KUKA KRL program: Up115.src, Up115.dat

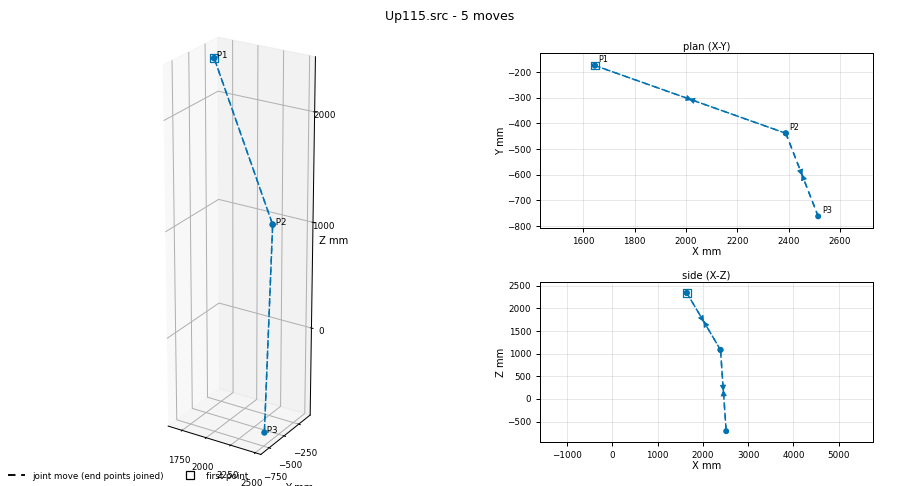
[picture p0: tool path of Up115.src, 5 of 5 moves have a stored position in this frame; points joined in program order, loops and branches not executed]
--- Up115.src ---
&ACCESS RV
&REL 2
&COMMENT Wartung Greifer 3 VW380
&PARAM DISKPATH = UPs
&PARAM TEMPLATE = C:\KRC\Roboter\Template\upvorgabe
&PARAM TPVW_VERSION = 8.1.8
&PARAM EDITMASK = Up999[1-999]
DEF UP115()
   ; FOLD UP Anfang;%{SE} %MKUKATPVW
   SPS_N=-1
   SPS_FERTIG=FALSE
   IF NOT CALLBYSELECT THEN
      INTERRUPT DECL 10 WHEN $CYCFLAG[254]==FALSE DO VW(#FB_STOP,TRUE)
      INTERRUPT ON 10
      INT10=TRUE
      VW_USR_R (#USR_INIT)
   ENDIF
   VW(#VW_INIT_UP,TRUE)
   ; ENDFOLD
   ;FOLD -- K2TUHR115425R01 Wartung Greifer VW380 -- ;%{PSE}%MKUKATPVW,%CVW_COM,%VCOMMENT,%P 1:Comment:, 2:K2TUHR115425R01 Wartung Greifer VW380
      ;FOLD {H}
         M_COMMENT("K2TUHR115425R01 Wartung Greifer VW380")
      ;ENDFOLD
   ;ENDFOLD
   ;FOLD PTP VB=100% VE=0% ACC=100% RobWzg=12 Base=0 SPSTrig=0[1/100s] P ;%{P}%MKUKATPVW,%CMOVE8,%VPTP,%P 1:1, 2: VB=, 3:100, 4:%, 5: VE=, 6:0, 7:%, 8: ACC=, 9:100, 10:%, 11: RobWzg=, 12:12, 13: Base=, 14:0, 15: SPSTrig=, 16:0, 17:[1/100s], 18: P, 19:1, 20:-1, 21:1
      ;FOLD 1: FB PSPS = EIN ;%{SE}%MKUKATPVW %CVW_SPS %VFBPSPS %P 2:FB PSPS = EIN,3:FBPSPS
      ;ENDFOLD
      ;FOLD 2: A23 = AUS ;%{SE}%MKUKATPVW %CVW_SPS %VBOASG %P 2:A23 = AUS,3:BOASG
      ;ENDFOLD
      ;FOLD 3: SPSMAKRO50 = EIN ;%{SE}%MKUKATPVW %CVW_SPS %VMAKRO %P 2:SPSMAKRO50 = EIN,3:MAKRO
      ;ENDFOLD
      ;FOLD 4: SPSMAKRO53 = EIN ;%{SE}%MKUKATPVW %CVW_SPS %VMAKRO %P 2:SPSMAKRO53 = EIN,3:MAKRO
      ;ENDFOLD
      ;FOLD 5: A42 = EIN ;%{SE}%MKUKATPVW %CVW_SPS %VBOASG %P 2:A42 = EIN,3:BOASG
      ;ENDFOLD
      ;FOLD 6: A43 = EIN ;%{SE}%MKUKATPVW %CVW_SPS %VBOASG %P 2:A43 = EIN,3:BOASG
      ;ENDFOLD
      ;FOLD 7: A44 = EIN ;%{SE}%MKUKATPVW %CVW_SPS %VBOASG %P 2:A44 = EIN,3:BOASG
      ;ENDFOLD
      ;FOLD 8: A45 = EIN ;%{SE}%MKUKATPVW %CVW_SPS %VBOASG %P 2:A45 = EIN,3:BOASG
      ;ENDFOLD
      ;FOLD 9: A47 = EIN ;%{SE}%MKUKATPVW %CVW_SPS %VBOASG %P 2:A47 = EIN,3:BOASG
      ;ENDFOLD
      ;FOLD 10: A49 = EIN ;%{SE}%MKUKATPVW %CVW_SPS %VBOASG %P 2:A49 = EIN,3:BOASG
      ;ENDFOLD
      ;FOLD 11: A52 = EIN ;%{SE}%MKUKATPVW %CVW_SPS %VBOASG %P 2:A52 = EIN,3:BOASG
      ;ENDFOLD
      ;FOLD 12: A54 = EIN ;%{SE}%MKUKATPVW %CVW_SPS %VBOASG %P 2:A54 = EIN,3:BOASG
      ;ENDFOLD
      ;FOLD 13: A75 = EIN ;%{SE}%MKUKATPVW %CVW_SPS %VBOASG %P 2:A75 = EIN,3:BOASG
      ;ENDFOLD
      ;FOLD 14: A76 = EIN ;%{SE}%MKUKATPVW %CVW_SPS %VBOASG %P 2:A76 = EIN,3:BOASG
      ;ENDFOLD
      ;FOLD 15: A79 = EIN ;%{SE}%MKUKATPVW %CVW_SPS %VBOASG %P 2:A79 = EIN,3:BOASG
      ;ENDFOLD
      ;FOLD 16: A80 = EIN ;%{SE}%MKUKATPVW %CVW_SPS %VBOASG %P 2:A80 = EIN,3:BOASG
      ;ENDFOLD
      ;FOLD 17: WARTE BIS M13 & M78 ;%{SE}%MKUKATPVW %CVW_SPS %VWBOASG %P 2:WARTE BIS M13 & M78,3:WBOASG
      ;ENDFOLD
      ;FOLD 18: F1 = EIN ;%{SE}%MKUKATPVW %CVW_SPS %VBOASG %P 2:F1 = EIN,3:BOASG
      ;ENDFOLD
      ;FOLD 19: F2 = EIN ;%{SE}%MKUKATPVW %CVW_SPS %VBOASG %P 2:F2 = EIN,3:BOASG
      ;ENDFOLD
      ;FOLD 20: SPSMAKRO342 = M13 ;%{SE}%MKUKATPVW %CVW_SPS %VMAKRO %P 2:SPSMAKRO342 = M13,3:MAKRO
      ;ENDFOLD
      ;FOLD 21: SPSMAKRO340 = EIN ;%{SE}%MKUKATPVW %CVW_SPS %VMAKRO %P 2:SPSMAKRO340 = EIN,3:MAKRO
      ;ENDFOLD
      ;FOLD 22: WARTE BIS M31 & M33 ;%{SE}%MKUKATPVW %CVW_SPS %VWBOASG %P 2:WARTE BIS M31 & M33,3:WBOASG
      ;ENDFOLD
      ;FOLD 23: WARTE BIS E23 ;%{SE}%MKUKATPVW %CVW_SPS %VWBOASG %P 2:WARTE BIS E23,3:WBOASG
      ;ENDFOLD
      ;FOLD 24: A23 = EIN ;%{SE}%MKUKATPVW %CVW_SPS %VBOASG %P 2:A23 = EIN,3:BOASG
      ;ENDFOLD
      ;FOLD 25: F841 = EIN ;%{SE}%MKUKATPVW %CVW_SPS %VBOASG %P 2:F841 = EIN,3:BOASG
      ;ENDFOLD
      ;FOLD 26: F842 = EIN ;%{SE}%MKUKATPVW %CVW_SPS %VBOASG %P 2:F842 = EIN,3:BOASG
      ;ENDFOLD
      ;FOLD 27: SPSMAKRO433 = EIN ;%{SE}%MKUKATPVW %CVW_SPS %VMAKRO %P 2:SPSMAKRO433 = EIN,3:MAKRO
      ;ENDFOLD
      ;FOLD 28: WARTE BIS !E547 & E548 & !E549 & E550 ;%{SE}%MKUKATPVW %CVW_SPS %VWBOASG %P 2:WARTE BIS !E547 & E548 & !E549 & E550,3:WBOASG
      ;ENDFOLD
      ;FOLD 29: FB PSPS = M13 & M30 & M31 & M33 & M78 ;%{SE}%MKUKATPVW %CVW_SPS %VFBPSPS %P 2:FB PSPS = M13 & M30 & M31 & M33 & M78,3:FBPSPS
      ;ENDFOLD
      ;FOLD {H}
         VW_MPARA_ACT=P1_D
         Act_P1 = P1
         Act_P2 = P1
         VW(#MPARA,TRUE)
         SPS_FERTIG=FALSE
         TRIGGER WHEN DISTANCE=1 DELAY=0 DO SPS_TRIG(1) PRIO=-1
         PTP P1
         $ADVANCE=1
         WAIT FOR SPS_FERTIG
      ;ENDFOLD
   ;ENDFOLD
   ;FOLD PTP VB=100% VE=100% ACC=100% RobWzg=12 Base=0 SPSTrig=0[1/100s] P ;%{P}%MKUKATPVW,%CMOVE8,%VPTP,%P 1:1, 2: VB=, 3:100, 4:%, 5: VE=, 6:100, 7:%, 8: ACC=, 9:100, 10:%, 11: RobWzg=, 12:12, 13: Base=, 14:0, 15: SPSTrig=, 16:0, 17:[1/100s], 18: P, 19:2, 20:-1, 21:2
      ;FOLD 1: FB PSPS = M13 & M30 & M31 & M33 & M78 ;%{SE}%MKUKATPVW %CVW_SPS %VFBPSPS %P 2:FB PSPS = M13 & M30 & M31 & M33 & M78,3:FBPSPS
      ;ENDFOLD
      ;FOLD {H}
         VW_MPARA_ACT=P2_D
         Act_P1 = P2
         Act_P2 = P2
         VW(#MPARA,TRUE)
         SPS_FERTIG=FALSE
         TRIGGER WHEN DISTANCE=1 DELAY=0 DO SPS_TRIG(10002) PRIO=-1
         PTP P2 C_PTP C_VEL
         $ADVANCE=1
      ;ENDFOLD
   ;ENDFOLD
   ;FOLD -- Wartungsposition Greifer VW380 -- ;%{PSE}%MKUKATPVW,%CVW_COM,%VCOMMENT,%P 1:Comment:, 2:Wartungsposition Greifer VW380
      ;FOLD {H}
         M_COMMENT("Wartungsposition Greifer VW380")
      ;ENDFOLD
   ;ENDFOLD
   ;FOLD PTP VB=100% VE=0% ACC=100% RobWzg=12 Base=0 SPSTrig=5[1/100s] P ;%{P}%MKUKATPVW,%CMOVE8,%VPTP,%P 1:1, 2: VB=, 3:100, 4:%, 5: VE=, 6:0, 7:%, 8: ACC=, 9:100, 10:%, 11: RobWzg=, 12:12, 13: Base=, 14:0, 15: SPSTrig=, 16:5, 17:[1/100s], 18: P, 19:3, 20:-1, 21:3
      ;FOLD 1: FB PSPS = EIN ;%{SE}%MKUKATPVW %CVW_SPS %VFBPSPS %P 2:FB PSPS = EIN,3:FBPSPS
      ;ENDFOLD
      ;FOLD 2: A23 = AUS ;%{SE}%MKUKATPVW %CVW_SPS %VBOASG %P 2:A23 = AUS,3:BOASG
      ;ENDFOLD
      ;FOLD 3: A17 = EIN ;%{SE}%MKUKATPVW %CVW_SPS %VBOASG %P 2:A17 = EIN,3:BOASG
      ;ENDFOLD
      ;FOLD 4: bin19 ( EIN ) = 3 ;%{SE}%MKUKATPVW %CVW_SPS %VARIASG %P 2:bin19 ( EIN ) = 3,3:ARIASG
      ;ENDFOLD
      ;FOLD 5: WARTE BIS E17 ;%{SE}%MKUKATPVW %CVW_SPS %VWBOASG %P 2:WARTE BIS E17,3:WBOASG
      ;ENDFOLD
      ;FOLD 6: A17 = AUS ;%{SE}%MKUKATPVW %CVW_SPS %VBOASG %P 2:A17 = AUS,3:BOASG
      ;ENDFOLD
      ;FOLD 7: bin19 ( EIN ) = 0 ;%{SE}%MKUKATPVW %CVW_SPS %VARIASG %P 2:bin19 ( EIN ) = 0,3:ARIASG
      ;ENDFOLD
      ;FOLD 8: WARTE BIS E23 ;%{SE}%MKUKATPVW %CVW_SPS %VWBOASG %P 2:WARTE BIS E23,3:WBOASG
      ;ENDFOLD
      ;FOLD 9: A23 = EIN ;%{SE}%MKUKATPVW %CVW_SPS %VBOASG %P 2:A23 = EIN,3:BOASG
      ;ENDFOLD
      ;FOLD 10: FB PSPS = M13 & M30 & M31 & M33 & M78 ;%{SE}%MKUKATPVW %CVW_SPS %VFBPSPS %P 2:FB PSPS = M13 & M30 & M31 & M33 & M78,3:FBPSPS
      ;ENDFOLD
      ;FOLD {H}
         VW_MPARA_ACT=P3_D
         Act_P1 = P3
         Act_P2 = P3
         VW(#MPARA,TRUE)
         SPS_FERTIG=FALSE
         TRIGGER WHEN DISTANCE=1 DELAY=-50 DO SPS_TRIG(3) PRIO=-1
         PTP P3
         $ADVANCE=1
         WAIT FOR SPS_FERTIG
      ;ENDFOLD
   ;ENDFOLD
   ;FOLD PTP VB=100% VE=100% ACC=100% RobWzg=12 Base=0 SPSTrig=0[1/100s] P ;%{P}%MKUKATPVW,%CMOVE8,%VPTP,%P 1:1, 2: VB=, 3:100, 4:%, 5: VE=, 6:100, 7:%, 8: ACC=, 9:100, 10:%, 11: RobWzg=, 12:12, 13: Base=, 14:0, 15: SPSTrig=, 16:0, 17:[1/100s], 18: P, 19:4, 20:-1, 21:4
      ;FOLD 1: FB PSPS = M13 & M30 & M31 & M33 & M78 ;%{SE}%MKUKATPVW %CVW_SPS %VFBPSPS %P 2:FB PSPS = M13 & M30 & M31 & M33 & M78,3:FBPSPS
      ;ENDFOLD
      ;FOLD {H}
         VW_MPARA_ACT=P4_D
         Act_P1 = P4
         Act_P2 = P4
         VW(#MPARA,TRUE)
         SPS_FERTIG=FALSE
         TRIGGER WHEN DISTANCE=1 DELAY=0 DO SPS_TRIG(10004) PRIO=-1
         PTP P4 C_PTP C_VEL
         $ADVANCE=1
      ;ENDFOLD
   ;ENDFOLD
   ;FOLD PTP VB=100% VE=0% ACC=100% RobWzg=12 Base=0 SPSTrig=0[1/100s] P ;%{P}%MKUKATPVW,%CMOVE8,%VPTP,%P 1:1, 2: VB=, 3:100, 4:%, 5: VE=, 6:0, 7:%, 8: ACC=, 9:100, 10:%, 11: RobWzg=, 12:12, 13: Base=, 14:0, 15: SPSTrig=, 16:0, 17:[1/100s], 18: P, 19:5, 20:-1, 21:5
      ;FOLD 1: FB PSPS = EIN ;%{SE}%MKUKATPVW %CVW_SPS %VFBPSPS %P 2:FB PSPS = EIN,3:FBPSPS
      ;ENDFOLD
      ;FOLD 2: A23 = AUS ;%{SE}%MKUKATPVW %CVW_SPS %VBOASG %P 2:A23 = AUS,3:BOASG
      ;ENDFOLD
      ;FOLD 3: WARTE BIS E23 ;%{SE}%MKUKATPVW %CVW_SPS %VWBOASG %P 2:WARTE BIS E23,3:WBOASG
      ;ENDFOLD
      ;FOLD 4: A23 = EIN ;%{SE}%MKUKATPVW %CVW_SPS %VBOASG %P 2:A23 = EIN,3:BOASG
      ;ENDFOLD
      ;FOLD 5: FB PSPS = M13 & M30 & M31 & M33 & M78 ;%{SE}%MKUKATPVW %CVW_SPS %VFBPSPS %P 2:FB PSPS = M13 & M30 & M31 & M33 & M78,3:FBPSPS
      ;ENDFOLD
      ;FOLD {H}
         VW_MPARA_ACT=P5_D
         Act_P1 = P5
         Act_P2 = P5
         VW(#MPARA,TRUE)
         SPS_FERTIG=FALSE
         TRIGGER WHEN DISTANCE=1 DELAY=0 DO SPS_TRIG(5) PRIO=-1
         PTP P5
         $ADVANCE=1
         WAIT FOR SPS_FERTIG
      ;ENDFOLD
   ;ENDFOLD
   ; FOLD ;%{H}
END
DEF SPS_TRIG(NO :IN)
   INT NO
   INT VW_STOP
   BOOL UES
   VW_STOP=$VW_PSPS_STOP
   IF NO>10000 THEN
      NO=NO-10000
      UES=TRUE
   ELSE
      UES=FALSE
   ENDIF
   ; FOLD ;%{H}
   IF ((VW_STOP B_AND 'B0001') > 0) THEN
      ;-- Trigger vorzeitig geschaltet (delay < 0) oder MStep
      IF (((VW_STOP B_AND 'B0110') > 0) AND ($MODE_OP<>#EX)) THEN
         ;-- MStep oder BCO Bewegung
         HALT
      ENDIF
   ENDIF
   ; ENDFOLD
   IF (SEARCH_END) THEN
      SEARCH_END = FALSE
      INTERRUPT OFF 39
   ENDIF
   SWITCH NO
      CASE 1
         ;FOLD SPS_TRIG1{H}
            VALCYCFL30=$CYCFLAG[254]
            $CYCFLAG[254]=(TRUE) AND $CYCFLAG[255] OR ($TIMER[61]<0)
            VW(#FB_CHECK,TRUE)
            $OUT[23] = FALSE
            SEL_RES=SELECT(#MAKRO,50,TRUE,,,,,FALSE)
            SEL_RES=SELECT(#MAKRO,53,TRUE,,,,,FALSE)
            $OUT[42] = TRUE
            $OUT[43] = TRUE
            $OUT[44] = TRUE
            $OUT[45] = TRUE
            $OUT[47] = TRUE
            $OUT[49] = TRUE
            $OUT[52] = TRUE
            $OUT[54] = TRUE
            $OUT[75] = TRUE
            $OUT[76] = TRUE
            $OUT[79] = TRUE
            $OUT[80] = TRUE
            $LOOP_MSG[]="M13 & M78"
            $LOOP_CONT=TRUE
            WAIT FOR ($CYCFLAG[13] AND $CYCFLAG[78]) OR (NOT $LOOP_CONT AND ($MODE_OP<>#EX))
            $LOOP_MSG[]="                                                                                                                                "
            $FLAG[1] = TRUE
            $FLAG[2] = TRUE
            SEL_RES=SELECT(#MAKRO,342,$CYCFLAG[13],,,,,FALSE)
            SEL_RES=SELECT(#MAKRO,340,TRUE,,,,,FALSE)
            $LOOP_MSG[]="M31 & M33"
            $LOOP_CONT=TRUE
            WAIT FOR ($CYCFLAG[31] AND $CYCFLAG[33]) OR (NOT $LOOP_CONT AND ($MODE_OP<>#EX))
            $LOOP_MSG[]="                                                                                                                                "
            $LOOP_MSG[]="E23"
            $LOOP_CONT=TRUE
            WAIT FOR ($IN[23]) OR (NOT $LOOP_CONT AND ($MODE_OP<>#EX))
            $LOOP_MSG[]="                                                                                                                                "
            $OUT[23] = TRUE
            $FLAG[841] = TRUE
            $FLAG[842] = TRUE
            SEL_RES=SELECT(#MAKRO,433,TRUE,,,,,FALSE)
            $LOOP_MSG[]="!E547 & E548 & !E549 & E550"
            $LOOP_CONT=TRUE
            WAIT FOR (NOT $IN[547] AND $IN[548] AND NOT $IN[549] AND $IN[550]) OR (NOT $LOOP_CONT AND ($MODE_OP<>#EX))
            $LOOP_MSG[]="                                                                                                                                "
            VALCYCFL30=$CYCFLAG[254]
            $CYCFLAG[254]=($CYCFLAG[13] AND $CYCFLAG[30] AND $CYCFLAG[31] AND $CYCFLAG[33] AND $CYCFLAG[78]) AND $CYCFLAG[255] OR ($TIMER[61]<0)
            VW(#FB_CHECK,TRUE)
         ;ENDFOLD
      CASE 2
         ;FOLD SPS_TRIG2{H}
            VALCYCFL30=$CYCFLAG[254]
            $CYCFLAG[254]=($CYCFLAG[13] AND $CYCFLAG[30] AND $CYCFLAG[31] AND $CYCFLAG[33] AND $CYCFLAG[78]) AND $CYCFLAG[255] OR ($TIMER[61]<0)
            VW(#FB_CHECK,TRUE)
         ;ENDFOLD
      CASE 3
         ;FOLD SPS_TRIG3{H}
            VALCYCFL30=$CYCFLAG[254]
            $CYCFLAG[254]=(TRUE) AND $CYCFLAG[255] OR ($TIMER[61]<0)
            VW(#FB_CHECK,TRUE)
            $OUT[23] = FALSE
            $OUT[17] = TRUE
            VW(#BINOUT,TRUE,19,3)
            $LOOP_MSG[]="E17"
            $LOOP_CONT=TRUE
            WAIT FOR ($IN[17]) OR (NOT $LOOP_CONT AND ($MODE_OP<>#EX))
            $LOOP_MSG[]="                                                                                                                                "
            $OUT[17] = FALSE
            VW(#BINOUT,TRUE,19,0)
            $LOOP_MSG[]="E23"
            $LOOP_CONT=TRUE
            WAIT FOR ($IN[23]) OR (NOT $LOOP_CONT AND ($MODE_OP<>#EX))
            $LOOP_MSG[]="                                                                                                                                "
            $OUT[23] = TRUE
            VALCYCFL30=$CYCFLAG[254]
            $CYCFLAG[254]=($CYCFLAG[13] AND $CYCFLAG[30] AND $CYCFLAG[31] AND $CYCFLAG[33] AND $CYCFLAG[78]) AND $CYCFLAG[255] OR ($TIMER[61]<0)
            VW(#FB_CHECK,TRUE)
         ;ENDFOLD
      CASE 4
         ;FOLD SPS_TRIG4{H}
            VALCYCFL30=$CYCFLAG[254]
            $CYCFLAG[254]=($CYCFLAG[13] AND $CYCFLAG[30] AND $CYCFLAG[31] AND $CYCFLAG[33] AND $CYCFLAG[78]) AND $CYCFLAG[255] OR ($TIMER[61]<0)
            VW(#FB_CHECK,TRUE)
         ;ENDFOLD
      CASE 5
         ;FOLD SPS_TRIG5{H}
            VALCYCFL30=$CYCFLAG[254]
            $CYCFLAG[254]=(TRUE) AND $CYCFLAG[255] OR ($TIMER[61]<0)
            VW(#FB_CHECK,TRUE)
            $OUT[23] = FALSE
            $LOOP_MSG[]="E23"
            $LOOP_CONT=TRUE
            WAIT FOR ($IN[23]) OR (NOT $LOOP_CONT AND ($MODE_OP<>#EX))
            $LOOP_MSG[]="                                                                                                                                "
            $OUT[23] = TRUE
            VALCYCFL30=$CYCFLAG[254]
            $CYCFLAG[254]=($CYCFLAG[13] AND $CYCFLAG[30] AND $CYCFLAG[31] AND $CYCFLAG[33] AND $CYCFLAG[78]) AND $CYCFLAG[255] OR ($TIMER[61]<0)
            VW(#FB_CHECK,TRUE)
         ;ENDFOLD
      CASE 6
         ;FOLD SPS_TRIG6{H}
         ;ENDFOLD
      CASE 7
         ;FOLD SPS_TRIG7{H}
         ;ENDFOLD
      CASE 8
         ;FOLD SPS_TRIG8{H}
         ;ENDFOLD
      CASE 9
         ;FOLD SPS_TRIG9{H}
         ;ENDFOLD
      CASE 10
         ;FOLD SPS_TRIG10{H}
         ;ENDFOLD
      CASE 11
         ;FOLD SPS_TRIG11{H}
         ;ENDFOLD
      CASE 12
         ;FOLD SPS_TRIG12{H}
         ;ENDFOLD
      CASE 13
         ;FOLD SPS_TRIG13{H}
         ;ENDFOLD
      CASE 14
         ;FOLD SPS_TRIG14{H}
         ;ENDFOLD
      CASE 15
         ;FOLD SPS_TRIG15{H}
         ;ENDFOLD
      CASE 16
         ;FOLD SPS_TRIG16{H}
         ;ENDFOLD
      CASE 17
         ;FOLD SPS_TRIG17{H}
         ;ENDFOLD
      CASE 18
         ;FOLD SPS_TRIG18{H}
         ;ENDFOLD
      CASE 19
         ;FOLD SPS_TRIG19{H}
         ;ENDFOLD
      CASE 20
         ;FOLD SPS_TRIG20{H}
         ;ENDFOLD
      CASE 21
         ;FOLD SPS_TRIG21{H}
         ;ENDFOLD
      CASE 22
         ;FOLD SPS_TRIG22{H}
         ;ENDFOLD
      CASE 23
         ;FOLD SPS_TRIG23{H}
         ;ENDFOLD
      CASE 24
         ;FOLD SPS_TRIG24{H}
         ;ENDFOLD
      CASE 25
         ;FOLD SPS_TRIG25{H}
         ;ENDFOLD
      CASE 26
         ;FOLD SPS_TRIG26{H}
         ;ENDFOLD
      CASE 27
         ;FOLD SPS_TRIG27{H}
         ;ENDFOLD
      CASE 28
         ;FOLD SPS_TRIG28{H}
         ;ENDFOLD
      CASE 29
         ;FOLD SPS_TRIG29{H}
         ;ENDFOLD
      CASE 30
         ;FOLD SPS_TRIG30{H}
         ;ENDFOLD
      CASE 31
         ;FOLD SPS_TRIG31{H}
         ;ENDFOLD
      CASE 32
         ;FOLD SPS_TRIG32{H}
         ;ENDFOLD
      CASE 33
         ;FOLD SPS_TRIG33{H}
         ;ENDFOLD
      CASE 34
         ;FOLD SPS_TRIG34{H}
         ;ENDFOLD
      CASE 35
         ;FOLD SPS_TRIG35{H}
         ;ENDFOLD
      CASE 36
         ;FOLD SPS_TRIG36{H}
         ;ENDFOLD
      CASE 37
         ;FOLD SPS_TRIG37{H}
         ;ENDFOLD
      CASE 38
         ;FOLD SPS_TRIG38{H}
         ;ENDFOLD
      CASE 39
         ;FOLD SPS_TRIG39{H}
         ;ENDFOLD
      CASE 40
         ;FOLD SPS_TRIG40{H}
         ;ENDFOLD
      CASE 41
         ;FOLD SPS_TRIG41{H}
         ;ENDFOLD
      CASE 42
         ;FOLD SPS_TRIG42{H}
         ;ENDFOLD
      CASE 43
         ;FOLD SPS_TRIG43{H}
         ;ENDFOLD
      CASE 44
         ;FOLD SPS_TRIG44{H}
         ;ENDFOLD
      CASE 45
         ;FOLD SPS_TRIG45{H}
         ;ENDFOLD
      CASE 46
         ;FOLD SPS_TRIG46{H}
         ;ENDFOLD
      CASE 47
         ;FOLD SPS_TRIG47{H}
         ;ENDFOLD
      CASE 48
         ;FOLD SPS_TRIG48{H}
         ;ENDFOLD
      CASE 49
         ;FOLD SPS_TRIG49{H}
         ;ENDFOLD
      CASE 50
         ;FOLD SPS_TRIG50{H}
         ;ENDFOLD
      CASE 51
         ;FOLD SPS_TRIG51{H}
         ;ENDFOLD
      CASE 52
         ;FOLD SPS_TRIG52{H}
         ;ENDFOLD
      CASE 53
         ;FOLD SPS_TRIG53{H}
         ;ENDFOLD
      CASE 54
         ;FOLD SPS_TRIG54{H}
         ;ENDFOLD
      CASE 55
         ;FOLD SPS_TRIG55{H}
         ;ENDFOLD
      CASE 56
         ;FOLD SPS_TRIG56{H}
         ;ENDFOLD
      CASE 57
         ;FOLD SPS_TRIG57{H}
         ;ENDFOLD
      CASE 58
         ;FOLD SPS_TRIG58{H}
         ;ENDFOLD
      CASE 59
         ;FOLD SPS_TRIG59{H}
         ;ENDFOLD
      CASE 60
         ;FOLD SPS_TRIG60{H}
         ;ENDFOLD
      CASE 61
         ;FOLD SPS_TRIG61{H}
         ;ENDFOLD
      CASE 62
         ;FOLD SPS_TRIG62{H}
         ;ENDFOLD
      CASE 63
         ;FOLD SPS_TRIG63{H}
         ;ENDFOLD
      CASE 64
         ;FOLD SPS_TRIG64{H}
         ;ENDFOLD
      CASE 65
         ;FOLD SPS_TRIG65{H}
         ;ENDFOLD
      CASE 66
         ;FOLD SPS_TRIG66{H}
         ;ENDFOLD
      CASE 67
         ;FOLD SPS_TRIG67{H}
         ;ENDFOLD
      CASE 68
         ;FOLD SPS_TRIG68{H}
         ;ENDFOLD
      CASE 69
         ;FOLD SPS_TRIG69{H}
         ;ENDFOLD
      CASE 70
         ;FOLD SPS_TRIG70{H}
         ;ENDFOLD
      CASE 71
         ;FOLD SPS_TRIG71{H}
         ;ENDFOLD
      CASE 72
         ;FOLD SPS_TRIG72{H}
         ;ENDFOLD
      CASE 73
         ;FOLD SPS_TRIG73{H}
         ;ENDFOLD
      CASE 74
         ;FOLD SPS_TRIG74{H}
         ;ENDFOLD
      CASE 75
         ;FOLD SPS_TRIG75{H}
         ;ENDFOLD
      CASE 76
         ;FOLD SPS_TRIG76{H}
         ;ENDFOLD
      CASE 77
         ;FOLD SPS_TRIG77{H}
         ;ENDFOLD
      CASE 78
         ;FOLD SPS_TRIG78{H}
         ;ENDFOLD
      CASE 79
         ;FOLD SPS_TRIG79{H}
         ;ENDFOLD
      CASE 80
         ;FOLD SPS_TRIG80{H}
         ;ENDFOLD
      CASE 81
         ;FOLD SPS_TRIG81{H}
         ;ENDFOLD
      CASE 82
         ;FOLD SPS_TRIG82{H}
         ;ENDFOLD
      CASE 83
         ;FOLD SPS_TRIG83{H}
         ;ENDFOLD
      CASE 84
         ;FOLD SPS_TRIG84{H}
         ;ENDFOLD
      CASE 85
         ;FOLD SPS_TRIG85{H}
         ;ENDFOLD
      CASE 86
         ;FOLD SPS_TRIG86{H}
         ;ENDFOLD
      CASE 87
         ;FOLD SPS_TRIG87{H}
         ;ENDFOLD
      CASE 88
         ;FOLD SPS_TRIG88{H}
         ;ENDFOLD
      CASE 89
         ;FOLD SPS_TRIG89{H}
         ;ENDFOLD
      CASE 90
         ;FOLD SPS_TRIG90{H}
         ;ENDFOLD
      CASE 91
         ;FOLD SPS_TRIG91{H}
         ;ENDFOLD
      CASE 92
         ;FOLD SPS_TRIG92{H}
         ;ENDFOLD
      CASE 93
         ;FOLD SPS_TRIG93{H}
         ;ENDFOLD
      CASE 94
         ;FOLD SPS_TRIG94{H}
         ;ENDFOLD
      CASE 95
         ;FOLD SPS_TRIG95{H}
         ;ENDFOLD
      CASE 96
         ;FOLD SPS_TRIG96{H}
         ;ENDFOLD
      CASE 97
         ;FOLD SPS_TRIG97{H}
         ;ENDFOLD
      CASE 98
         ;FOLD SPS_TRIG98{H}
         ;ENDFOLD
      CASE 99
         ;FOLD SPS_TRIG99{H}
         ;ENDFOLD
      CASE 100
         ;FOLD SPS_TRIG100{H}
         ;ENDFOLD
      CASE 101
         ;FOLD SPS_TRIG101{H}
         ;ENDFOLD
      CASE 102
         ;FOLD SPS_TRIG102{H}
         ;ENDFOLD
      CASE 103
         ;FOLD SPS_TRIG103{H}
         ;ENDFOLD
      CASE 104
         ;FOLD SPS_TRIG104{H}
         ;ENDFOLD
      CASE 105
         ;FOLD SPS_TRIG105{H}
         ;ENDFOLD
      CASE 106
         ;FOLD SPS_TRIG106{H}
         ;ENDFOLD
   DEFAULT
   ENDSWITCH
   ; FOLD ;%{H}
   IF ($MODE_OP<>#EX) THEN
      ;-- Trigger erst nach Wiederanstart geschaltet --
      IF ((((VW_STOP B_AND 'B10010') >0) AND ((VW_STOP B_AND 'B0001')<=0))) THEN
         ;-- MStep Bewegung --
         HALT
      ENDIF
   ENDIF
   ; ENDFOLD
   IF NOT UES THEN
      SPS_FERTIG=TRUE
   ENDIF
END
; ENDFOLD

--- Up115.dat ---
&ACCESS RV
&REL 2
&COMMENT Wartung Greifer 3 VW380
&PARAM DISKPATH = UPs
&PARAM TEMPLATE = C:\KRC\Roboter\Template\upvorgabe
&PARAM TPVW_VERSION = 8.1.8
&PARAM EDITMASK = Up999[1-999]
DEFDAT UP115
; FOLD ;%{H} %MKUKATPVW
; ENDFOLD
; interface to basic routines
 EXT  BAS (BAS_COMMAND  :IN,REAL  :IN )
; interface to VW-standard routines
EXT VW (VW_COMMAND:IN, BOOL: IN, REAL:IN, REAL:IN, REAL:IN, REAL:IN, BOOL :IN, E6POS :IN )
; interface to VW_USER - Call
EXT  VW_USER (VW_USER_CMD :IN,INT :IN,REAL  :IN,REAL  :IN,REAL  :IN,REAL  :IN,REAL  :IN,REAL  :IN,BOOL  :IN )
EXT  VW_USR_R (VW_USER_CMD :IN,INT :IN,REAL  :IN,REAL  :IN,REAL  :IN,REAL  :IN,REAL  :IN,REAL  :IN,BOOL  :IN )
EXT  IBGN (IBGN_COMMAND  :IN,BOOL  :IN,REAL  :IN,REAL  :IN,BOOL  :IN,E6POS  :OUT )
; interface select routine
EXTFCT INT  SELECT (SUBTYPE  :IN,INT  :IN,BOOL  :IN,ARI_TYP  :IN,INT  :IN,BOOL_TYP  :IN,INT  :IN,BOOL  :IN)
INT VW_NEXT_FREE = 6
INT VW_NFREE_SPS = 6
INT VW_MAX_SPS = 106
DECL VW_MPARA_TYP P1_D = {TOOL_NO 12,BASE_NO 0,VB 100,VE 0,ACC 100,TRG_TIME 0,MOVE_TYPE #PTP_MOTION}
DECL E6POS P1 = {X 1644.416, Y -174.6792, Z 2340.625, A 0.01452038, B 29.99903, C -90.35256, S 2, T 42 , E1 0.0, E2 0.0, E3 0.0, E4 0.0, E5 0.0, E6 0.0}
DECL VW_MPARA_TYP P2_D = {TOOL_NO 12,BASE_NO 0,VB 100,VE 100,ACC 100,TRG_TIME 0,MOVE_TYPE #PTP_MOTION}
DECL E6POS P2 = {X 2388.61, Y -438.7298, Z 1083.309, A -2.522015, B 49.97304, C -8.240117, S 2, T 42 , E1 0.0, E2 0.0, E3 0.0, E4 0.0, E5 0.0, E6 0.0}
DECL VW_MPARA_TYP P3_D = {TOOL_NO 12,BASE_NO 0,VB 100,VE 0,ACC 100,TRG_TIME 5,MOVE_TYPE #PTP_MOTION}
DECL E6POS P3 = {X 2514.471, Y -762.2805, Z -712.819, A 4.802316, B 87.00743, C 6.317693, S 2, T 42 , E1 0.0, E2 0.0, E3 0.0, E4 0.0, E5 0.0, E6 0.0}
DECL VW_MPARA_TYP P4_D = {TOOL_NO 12,BASE_NO 0,VB 100,VE 100,ACC 100,TRG_TIME 0,MOVE_TYPE #PTP_MOTION}
DECL E6POS P4 = {X 2388.61, Y -438.7298, Z 1083.309, A -2.522015, B 49.97304, C -8.240117, S 2, T 42 , E1 0.0, E2 0.0, E3 0.0, E4 0.0, E5 0.0, E6 0.0}
DECL VW_MPARA_TYP P5_D = {TOOL_NO 12,BASE_NO 0,VB 100,VE 0,ACC 100,TRG_TIME 0,MOVE_TYPE #PTP_MOTION}
DECL E6POS P5 = {X 1644.416, Y -174.6797, Z 2340.624, A 0.01450222, B 29.99903, C -90.35255, S 2, T 42 , E1 0.0, E2 0.0, E3 0.0, E4 0.0, E5 0.0, E6 0.0}
ENDDAT
